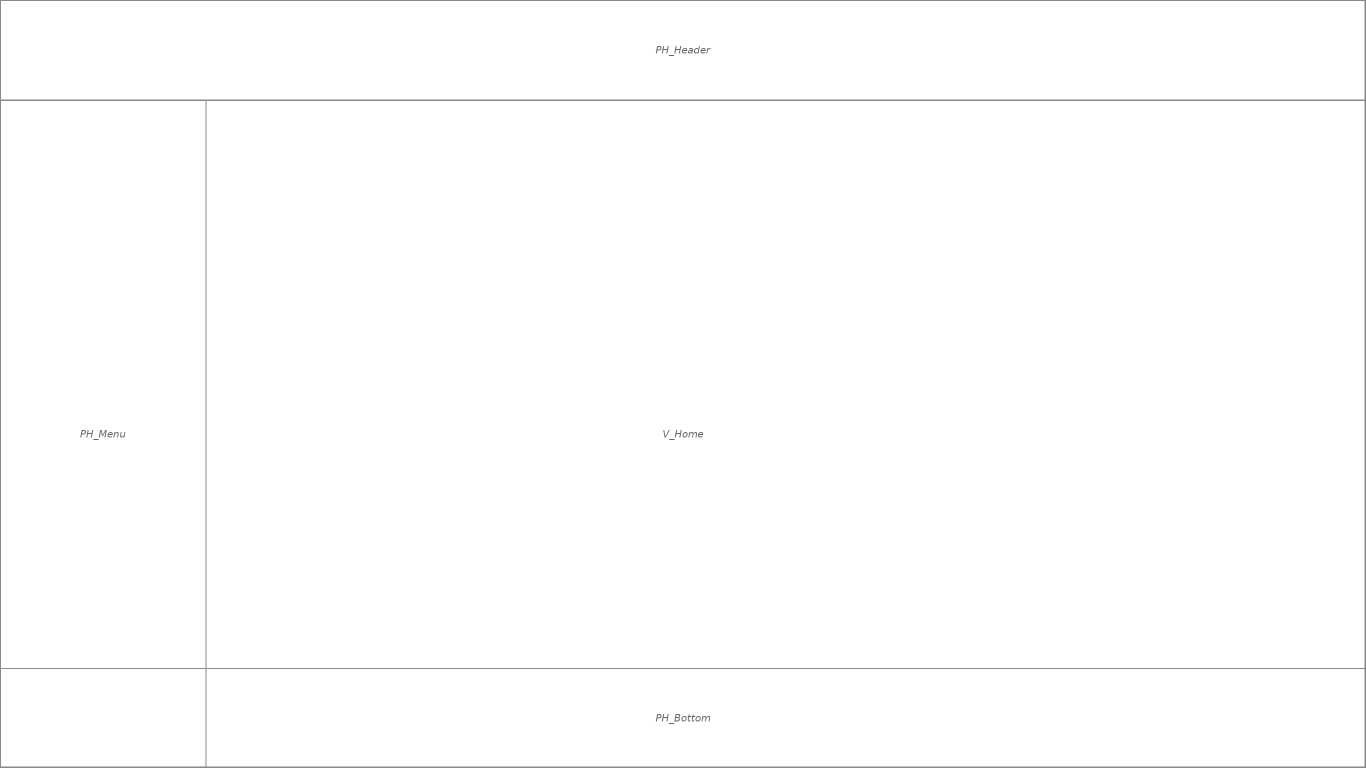
VISUALIZATION Visualization  // 1366x768
    Frame (0,0 1366x100)
        shows PH_Header(iFrameNumber := GVL_HMI.iFrameNumber, bMenu := GVL_HMI.bMenu, wButton := GVL_HMI.wButton)
    Frame (0,100 1366x668), frame switch variable: GVL_HMI.iFrameNumber
        shows V_Home(bKillProcess := P_CloseTcHmiExe.bKillProcess, sImageOsName := P_ControllerInfo.stDevIdent.strImageOsName)
        shows V_EventsHistoricalSimple()
        shows V_info()
        shows V_Users()
        shows V_Settings()
        shows V_FileDialog()
        shows V_Table(arrTable := P_Table.arrTable, iColumn := P_Table.iColumn, iLine := P_Table.iLine, iValue := P_Table.iValue, iSetValue := P_Table.iSetValue, bSet := P_Table.bSetNewValue)
        shows V_Trend(arrHistogram := P_Table.arrHistogram, bShow := P_Table.bRotate)
        shows V_Option4()
        shows V_Option5()
        shows V_Option6()
    Frame (0,100 206x668), invisible if: NOT GVL_HMI.bMenu
        shows PH_Menu(bMain1 := GVL_HMI.bMain1, bMain2 := GVL_HMI.bMain2, iFrameNumber := GVL_HMI.iFrameNumber, udiFOntColor1 := GVL_HMI.udiFOntColor1, udiFontColor2 := GVL_HMI.udiFOntColor2)
    Frame (0,668 1366x100), invisible if: GVL_HMI.iFrameNumber=1
        shows PH_Bottom(bReset := GVL_HMI.bReset, arrEventVisu := GVL_EHS.arrEventVisu)
END_VISUALIZATION

(* stored: Version 1.1.0.1, ProductVersion 3.1.4024.3
   Visu Visualization: Id {ae93cdc2-e691-4410-a6b4-92f7a89a2e7a} *)
